(* PLC project  *)

CONFIGURATION Empty_Module_28
END_CONFIGURATION
